SUBAPPLICATION StringValue_TO_INI (* String-VT-Wert einlesen und in INI speichern (generisch). *)
  (* Standard: 61499-2 *)
  (* Version 1.0, 2026-09-09, Franz Höpfinger, Meisterschulen am Ostbahnhof, Ausgelagert aus Uebung_012k_sub zur Wiederverwendung. *)
  PACKAGE MyLib::sys;
  IMPORT isobus::UT::Q::const::IDs::ID_NULL;
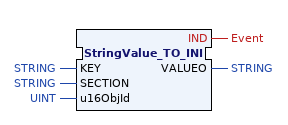
  EVENT_OUTPUT
    IND;
  END_EVENT
  VAR_INPUT
    KEY : STRING; (* Key name. *)
    SECTION : STRING; (* Section name. *)
    u16ObjId : UINT := ID_NULL;
  END_VAR
  VAR_OUTPUT
    VALUEO : STRING;
  END_VAR
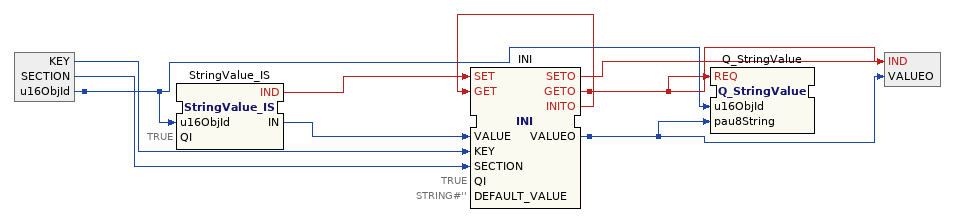
  FBS
    StringValue_IS : isobus::UT::io::StringValue::StringValue_IS(QI := TRUE);
    INI : eclipse4diac::storage::INI(QI := TRUE, DEFAULT_VALUE := STRING#'');
    Q_StringValue : isobus::UT::Q::Q_StringValue;
  END_FBS
  EVENT_CONNECTIONS
    StringValue_IS.IND TO INI.SET;
    INI.SETO TO IND;
    INI.GETO TO Q_StringValue.REQ;
    INI.GETO TO IND;
    INI.INITO TO INI.GET;
  END_CONNECTIONS
  DATA_CONNECTIONS
    StringValue_IS.IN TO INI.VALUE;
    u16ObjId TO Q_StringValue.u16ObjId;
    KEY TO INI.KEY;
    INI.VALUEO TO Q_StringValue.pau8String;
    INI.VALUEO TO VALUEO;
    u16ObjId TO StringValue_IS.u16ObjId;
    SECTION TO INI.SECTION;
  END_CONNECTIONS
END_SUBAPPLICATION
